// TIA Portal V19 export
DATA_BLOCK "RTE_405_DB"   // DB405
{ S7_Optimized_Access := 'TRUE' }
AUTHOR : HGS
FAMILY : SERVICE
// stored: AutoNumber false, MemoryReserve 0
   VAR RETAIN
      HMI : Struct   // HMI data structure
         ROUTE_ID : Int := 22;   // Route number running
         STEP_NUMBER : Int;   // Current step number
         STEP_IDENT_TEXT_NUMBER : Int;   // Sequence step text number
         STEP_VALUE : Int;   // Value of current step data (Time/weight/volume/cycles etc)
         STEP_VALUE_DIMENSION : Int;   // Step value dimension (0 = None/1=Seconds/2=Minutes/3=Kg/4=Litres)
         ERROR_TEXT_NUMBER : Int;   // Route start error message number for HMI
         INF_TEXT_NUMBER : Int;   // Route information message number for HMI
         STEP_VALUE_REAL : Real := 0.0;   // Value of current step data (Time/weight/volume/cycles etc) REAL
         NEXT_STEP : Int;   // Next step number
         FAULT : Bool := TRUE;   // Route fault active flag
         NOT_AVAILABLE : Bool;   // Route not available flag
         RUNNING : Bool;   // Route running flag
         TIMER_HELD : Bool;   // Timer held flag
         SEQUENCE_HELD : Bool;   // Sequence held flag
         SEQUENCE_ABORTED : Bool;   // Sequence aborted flag
         Spare_20_6 : Bool;   // Spare
         Spare_20_7 : Bool;   // Spare
         SEQ_RUNNING_ONS_MEM : Bool;   // Spare
         SEQ_RUNNING_ONS : Bool;   // Spare
         SEQ_STOPPED_ONS_MEM : Bool;   // Spare
         SEQ_STOPPED_ONS : Bool;   // Spare
         Spare_21_4 : Bool;   // Spare
         Spare_21_5 : Bool;   // Spare
         Spare_21_6 : Bool;   // Spare
         Route_Healthy : Bool;   // Route Healthy
      END_STRUCT;
      CONTROL : Struct
         MESSAGE_TIME : Int;   // Sequence error message elapsed time
         ERROR_MESSAGE_MEM : Int;   // Sequence error message memory
         STEP_TIME : DInt := DINT#14838493;   // Time sequence has been on current step
      END_STRUCT;
      FLAGS : Struct
         Device_Fault : Bool := TRUE;   // Circuit Device in Fault
         Process_Fault : Bool;   // Circuit Process Fault
         Step_Value_Done : Bool := TRUE;   // Current step value decremented to zero
         Sequence_Ended : Bool;   // Sequence complete flag
         Step_Change : Bool;   // Step changed flag
         Step_Count_Enable : Bool := TRUE;   // Enable step count down
         STEP_0 : Bool := TRUE;   // Spare
         STEP_END : Bool;   // Spare
         STEP_1_0 : Bool;   // Step 1.0 - Set Route
         STEP_2_0 : Bool;   // Step 2.0 - Heating
         STEP_3_0 : Bool;   // Step 3.0 - Sterilising Time
         STEP_4_0 : Bool;   // Step 4.0 - Cooling
         STEP_5_0 : Bool;   // Step 5.0 - Cooling Temp Check
         STEP_6_0 : Bool;   // Step 6.0 - EOL Barrier ON
         Sequence_Start : Bool;   // Sequence Start Signal
         STEP_7_0 : Bool;   // Step 7.0 - Inlet Barrier ON
         STEP_8_0 : Bool;   // Step 8.0 - Set Sterile Status
         ENCYL_3 : Bool;   // ENAHVCY Cycle 3 V12/13/21
         _2_2 : Bool;   // Spare
         _2_3 : Bool;   // Spare
         Sterile : Bool;   // Sterile Status Bit
         Production_Req : Bool;   // Goto Production
         _2_6 : Bool;   // Spare
         _2_7 : Bool;   // Spare
         _3 : Byte;   // Spare
         _4 : Byte;   // Spare
         _5 : Byte;   // Spare
         _6 : Byte;   // Spare
         _7 : Byte;   // Spare
         _8 : Byte;   // Spare
         _9 : Byte;   // Spare
      END_STRUCT;
      HMI_CMD : Struct   // Polygon Custard > Gemini CIP Commands
         Timer_Hold : Bool;   // Timer Hold
         Timer_Release : Bool;   // Timer Release
         Hold : Bool;   // Route hold
         Continue : Bool;   // Route continue
         Abort : Bool;   // Route abort
         Start : Bool;   // Route Start
         _0_6 : Bool;   // Spare Flag
         _0_7 : Bool;   // Spare Flag
         Timer_Hold_Available : Bool;
         Timer_Release_Available : Bool;
         Hold_Available : Bool;   // Enable HMI Hold pb
         Continue_Available : Bool;   // Enable HMI Resume pb
         Abort_Available : Bool;   // Enable HMI Abort pb
         Start_Available : Bool;   // Enable HMI Start pb
         _1_6 : Bool;   // Spare Flag
         _1_7 : Bool;   // Spare Flag
      END_STRUCT;
      PARAMETERS : Struct   // Sequence Parameters
         PARAM_01 : Int := 1800;   // Sequence Parameter - (T6) SIP Time
         PARAM_02 : Int := 240;   // Sequence Parameter - (T7) SIP Drain Down Time
         PARAM_03 : Int := 240;   // Sequence Parameter - (T13) EOL Barrier Cycle 1(V12/14/21 ON)
         PARAM_04 : Int := 5;   // Sequence Parameter - (T14) EOL Barrier Cycle 2(V12 ON)
         PARAM_05 : Int := 5;   // Sequence Parameter - (T15) EOL Barrier Cycle 3(V12/14 ON)
         PARAM_03_Act : DInt := DINT#152476;   // Sequence Parameter - (T13) EOL Barrier Cycle 1(V12/14/21 ON) Actual
         PARAM_04_Act : DInt;   // Sequence Parameter - (T14) EOL Barrier Cycle 2(V12 ON) Actual
         PARAM_05_Act : DInt;   // Sequence Parameter - (T15) EOL Barrier Cycle 3(V12/14 ON) Actual
      END_STRUCT;
   END_VAR
BEGIN
END_DATA_BLOCK
